// Generated by SQL Query Editor
TYPE ST_MachineParameter :
STRUCT
	iParameters_Index	: INT;
	wsTag_Name			: WSTRING(255);
	iStation			: INT;
	wsParameters_Unit	: WSTRING(50);
	iPackTagID			: INT;
	wsParameters_Value	: WSTRING(255);
	eDataType			: E_DB_DataType;
END_STRUCT
END_TYPE


//SQL Command
(*
SELECT          Global_Machine_Parameters.Parameters_Index, 
				Global_Machine_Parameters.Parameters_Name, 
				Global_Machine_Parameters.Station, 
				Global_Machine_Parameters.Parameters_Unit,
                Global_Machine_Parameters.PackTagID, 
				Global_Machine_Parameters_Value.Parameters_Value
FROM            Global_Machine_Parameters_Value INNER JOIN
                Global_Machine_Parameters ON 
                Global_Machine_Parameters_Value.Parameters_Index = Global_Machine_Parameters.Parameters_Index
ORDER BY Global_Machine_Parameters.Parameters_Index
*)

(* stored: Version 1.1.0.1, ProductVersion 3.1.4024.11
   DUT ST_MachineParameter: Id {b49474ae-4465-4800-801e-fcf277cb5b82} *)
